FUNCTION_BLOCK FB_Component_Servo IMPLEMENTS I_Component
VAR_INPUT
	sName				: STRING[50];			
	tTimeout			: TIME := T#0MS;
	
	uMaxRPMservo		: INT;		// value set in servo drive ( == RPM before gears!!)
	rGearRatio			: REAL;
END_VAR

VAR_IN_OUT
	bRTO				: BOOL;
	bEnableDrive		: BOOL;
	bResetDrive			: BOOL;
	uAnalogOut			: INT;
	
	(*bSetCounterDone		: BOOL;
	dCount				: DINT;
	bSetCounter			: BOOL;
	dSetCounterValue	: DINT;*)
END_VAR

VAR_OUTPUT
	
	bEnabled			: BOOL;
	eState				: E_State 				:= E_State.DISABLED;
	eServoState			: E_ServoStateMachine 	:= E_ServoStateMachine.IDLE;
	sStatusText 		: STRING[100];
END_VAR

VAR
	tTimeoutTimer		: TON;
	eLastState			: E_State;
	
	uInitialRPM			: INT;
	uTargetRPM			: INT;
	uCurrRPM			: INT;
	uRPMlimit			: INT := 0;
	uAcceleration		: INT := 0;		// RPM/s
	bDirection			: BOOL;			// FALSE = CW, TRUE = CCW
	tAccelerationTimer	: TON;
END_VAR

VAR CONSTANT
	DISABLED			: E_State := E_State.DISABLED;
	READY				: E_State := E_State.READY;
	BUSY				: E_State := E_State.BUSY;
	DONE				: E_State := E_State.DONE;
	HALTED				: E_State := E_State.HALTED;
	TIMEOUT				: E_State := E_State.TIMEOUT;
	
	IDLE       			: E_ServoStateMachine := E_ServoStateMachine.IDLE;
	HOMING     			: E_ServoStateMachine := E_ServoStateMachine.HOMING;
	HOMED      			: E_ServoStateMachine := E_ServoStateMachine.HOMED;
	RAMPUP     			: E_ServoStateMachine := E_ServoStateMachine.RAMPUP;
	HOLD       			: E_ServoStateMachine := E_ServoStateMachine.HOLD;
	RAMPDOWN   			: E_ServoStateMachine := E_ServoStateMachine.RAMPDOWN;
	FAULT      			: E_ServoStateMachine := E_ServoStateMachine.FAULT;
END_VAR

tTimeoutTimer.PT		:= tTimeout;
tAccelerationTimer.PT 	:= T#30M;

uCurrRPM := REAL_TO_INT((((INT_TO_REAL(ABS(uAnalogOut))/32767)) * uMaxRPMservo) / rGearRatio);

CASE eState OF
	DISABLED: 	sStatusText := '';
	READY: 		sStatusText := '';
	BUSY: 		sStatusText := '';
				CASE eServoState OF
					IDLE:
						IF bEnableDrive AND NOT bRTO THEN
							M_Reset();
						END_IF
						tAccelerationTimer(IN := FALSE);
					HOMING:
						eServoState := HOMING; // placeholder
					HOMED:
						eServoState := HOMED; // placeholder
					RAMPUP:
						tAccelerationTimer(IN := TRUE);
						IF uCurrRPM = uTargetRPM THEN
							eServoState := HOLD;
						ELSE
							uCurrRPM := M_CalculateRPM(uTargetRPM := uTargetRPM, uInitialRPM := uInitialRPM, rElapsedTime := tAccelerationTimer.ET);
						END_IF
					HOLD:
						eServoState := HOLD; // placeholder
					RAMPDOWN:
						tAccelerationTimer(IN := TRUE);
						IF uCurrRPM = uTargetRPM THEN
							eServoState := HOLD;
						ELSE
							uCurrRPM := M_CalculateRPM(uTargetRPM := uTargetRPM, uInitialRPM := uInitialRPM, rElapsedTime := tAccelerationTimer.ET);
						END_IF
					FAULT:
						eServoState := FAULT;
				END_CASE
	TIMEOUT:	sStatusText := '';
	DONE:		sStatusText := '';
	HALTED:		sStatusText := '';
END_CASE


// uCurrRPM := REAL_TO_INT((((INT_TO_REAL(ABS(uAnalogOut))/32767)) * uMaxRPM) / rGearRatio);

METHOD M_CalculateRPM : INT
VAR_INPUT
	uTargetRPM  	: INT;
	uInitialRPM		: INT;
	rElapsedTime	: TIME;
END_VAR

VAR
	uRPMdiff		: INT; // rpm to add to initial rpm
END_VAR
uRPMdiff := REAL_TO_INT((TIME_TO_REAL(rElapsedTime) / 100) * uAcceleration);

CASE eServoState OF
	RAMPUP:
		M_CalculateRPM := SEL((uInitialRPM + uRPMdiff) >= uTargetRPM, (uInitialRPM + uRPMdiff), uTargetRPM);
	RAMPDOWN:
		M_CalculateRPM := SEL((uInitialRPM - uRPMdiff) <= uTargetRPM, (uInitialRPM - uRPMdiff), uTargetRPM);
END_CASE
END_METHOD

{warning 'add method implementation '}
METHOD M_Disable : BOOL
END_METHOD

{warning 'add method implementation '}
METHOD M_Enable : BOOL
END_METHOD

{warning 'add method implementation '}
METHOD M_Halt : BOOL
END_METHOD

{warning 'add method implementation '}
METHOD M_Reset : BOOL
END_METHOD

{warning 'add method implementation '}
METHOD M_Resume : BOOL
END_METHOD

METHOD M_SetAcceleration : BOOL
VAR_INPUT
	uRPMperSec : INT;
END_VAR
uAcceleration := SEL(uRPMperSec >= 500, uRPMperSec, 500);
END_METHOD

METHOD M_SetRPMlimit : BOOL
VAR_INPUT
	RPM 				: INT;
	uMaxRPMafterGears	: INT;
END_VAR
uMaxRPMafterGears 	:= REAL_TO_INT(INT_TO_REAL(uMaxRPMservo / rGearRatio));
uRPMlimit 			:= SEL(RPM >= uMaxRPMafterGears, RPM, uMaxRPMafterGears);
END_METHOD

METHOD M_SetTargetRPM : BOOL
VAR_INPUT
	RPM : INT;
END_VAR
IF eState = READY OR eState = BUSY THEN
	tAccelerationTimer(IN := FALSE);	// reset the timer
	IF uTargetRPM > uCurrRPM THEN
		eServoState := RAMPUP;
	ELSIF uTargetRPM < uCurrRPM THEN
		eServoState := RAMPDOWN;
	ELSE
		eServoState := HOLD;
	END_IF
	uInitialRPM	:= uCurrRPM;
	uTargetRPM 	:= SEL(RPM >= uRPMlimit, RPM, uRPMlimit);
END_IF;
END_METHOD

{warning 'add method implementation '}
METHOD M_Stop : BOOL
END_METHOD

END_FUNCTION_BLOCK

(* stored: Version 1.1.0.1, ProductVersion 3.1.4024.15
   POU FB_Component_Servo: Id {ffbd4ec0-98dd-4a8f-a9df-1ac783cdf63e}, SpecialFunc None
   Method M_CalculateRPM: Id {e71f719e-2a3d-4a51-8521-69420927a634}
   Method M_Disable: Id {1162f5c2-57a8-43b1-b001-97555c860349}
   Method M_Enable: Id {0b6461d7-9c72-4480-b0c7-4f04c006cb47}
   Method M_Halt: Id {4d90e9ea-c4c4-4688-bc3f-883478b503e7}
   Method M_Reset: Id {65588943-8c9f-4d08-9d58-f2d9bbca6093}
   Method M_Resume: Id {0ef55e00-fae7-4950-b428-9b3b80a98729}
   Method M_SetAcceleration: Id {78d30c80-f4c9-4891-8275-0303f69aba9b}
   Method M_SetRPMlimit: Id {8fa04868-0f1b-4aad-a5f3-d61560b4199d}
   Method M_SetTargetRPM: Id {77e80cf1-83a2-41c2-a47e-e1c57835fa8e}
   Method M_Stop: Id {4937a094-2c8a-434b-9e0b-55e8bd81c853} *)
